(*********************************** G.D S.p.A. - Technical Department ***********************************
============= PROGRAM INFO ============
FOLDER:             TBD
MACHINES INVOLVED:  TBD 

============= DESCRIPTION =============
csp main interface program

============= REVISIONS ===============
Date		Version	 	Author      	Description             
----------	-------		------------  	--------------------------------------------
2019/09/27 	0000.00	 	M.Grasso		Creation of the PRG

**********************************************************************************************************)
PROGRAM _csp_case_closing_normal
VAR
END_VAR

(* CASE *)
	(* CLOSING *)
		(* OS *)
		csp_case_closing_os();
	
		(* LS *)
		csp_case_closing_ls();

END_PROGRAM

(* stored: Version 1.1.0.1, ProductVersion 3.1.4022.12
   POU _csp_case_closing_normal: Id {701a2a2d-ecec-41bb-a331-a3bb5823b6a8}, SpecialFunc None *)
